// TIA Portal V16 export
// export: Created 2024-09-05T17:39:24.436191Z, ExportSetting WithDefaults, DisplayName Totally Integrated Automation Portal, DisplayVersion V16 Update 6, DisplayName TIA Portal Version Control Interface, DisplayVersion V16 Update 2, DisplayName TIA Portal Openness, DisplayVersion V16 Update 6, DisplayName STEP 7 Professional, DisplayVersion V16 Update 6, DisplayName STEP 7 Safety, DisplayVersion V16, DisplayName WinCC Advanced, DisplayVersion V16 Update 6
FUNCTION "Concatenate_STRING" : Void   // FC2010, LAD
{ S7_Optimized_Access := 'TRUE' }
VERSION : 0.1
// stored: AutoNumber false, IsIECCheckEnabled false, SetENOAutomatically false, UDAEnableTagReadback false
   VAR_INPUT
      DMC_SAP_REF : Array[1..10] of String[25];
   END_VAR
   VAR_OUTPUT
      String_empty : Bool;
   END_VAR
   VAR_IN_OUT
      DMC_SAP_REf_WSTRING : WString;
   END_VAR
   VAR_TEMP
      concatenate : String;
      Convert : WString;
   END_VAR
   VAR CONSTANT
      Template_string_empty : String := ';;;;;;;;;';
   END_VAR
BEGIN

REGION Network 1 (SCL): Concatenate function
       #concatenate := CONCAT(IN1 := #DMC_SAP_REF[1], IN2 := ';');
       #concatenate := CONCAT(IN1 := #concatenate, IN2 := #DMC_SAP_REF[2]);
       #concatenate := CONCAT(IN1 := #concatenate, IN2 := ';');
       #concatenate := CONCAT(IN1 := #concatenate, IN2 := #DMC_SAP_REF[3]);
       #concatenate := CONCAT(IN1 := #concatenate, IN2 := ';');
       #concatenate := CONCAT(IN1 := #concatenate, IN2 := #DMC_SAP_REF[4]);
       #concatenate := CONCAT(IN1 := #concatenate, IN2 := ';');
       #concatenate := CONCAT(IN1 := #concatenate, IN2 := #DMC_SAP_REF[5]);
       #concatenate := CONCAT(IN1 := #concatenate, IN2 := ';');
       #concatenate := CONCAT(IN1 := #concatenate, IN2 := #DMC_SAP_REF[6]);
       #concatenate := CONCAT(IN1 := #concatenate, IN2 := ';');
       #concatenate := CONCAT(IN1 := #concatenate, IN2 := #DMC_SAP_REF[7]);
       #concatenate := CONCAT(IN1 := #concatenate, IN2 := ';');
       #concatenate := CONCAT(IN1 := #concatenate, IN2 := #DMC_SAP_REF[8]);
       #concatenate := CONCAT(IN1 := #concatenate, IN2 := ';');
       #concatenate := CONCAT(IN1 := #concatenate, IN2 := #DMC_SAP_REF[9]);
       #concatenate := CONCAT(IN1 := #concatenate, IN2 := ';');
       #concatenate := CONCAT(IN1 := #concatenate, IN2 := #DMC_SAP_REF[10]);
END_REGION

REGION Network 2
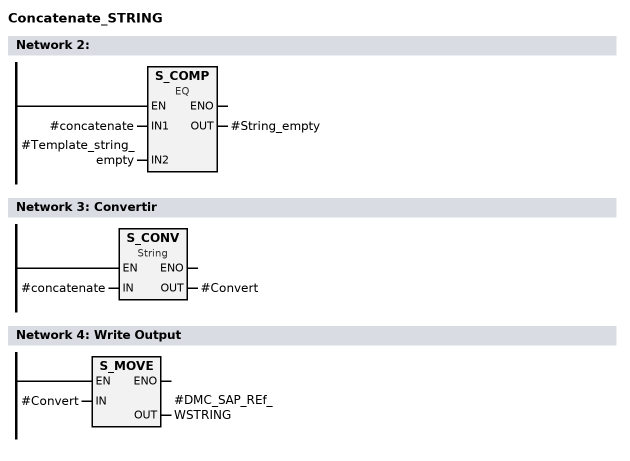
   RUNG wire#powerrail
      { S7_Templates := "[relation := EQ, src_type := String]" } S_COMP(IN1 := #concatenate, IN2 := #Template_string_empty, OUT => #String_empty)
   END_RUNG
   // the same network as SCL:
   S_COMP(IN1 := #concatenate, IN2 := #Template_string_empty, OUT => #String_empty);
END_REGION

REGION Network 3: Convertir
   RUNG wire#powerrail
      { S7_Templates := "[src_type := String, dest_type := WString]" } S_CONV(IN := #concatenate, OUT => #Convert)
   END_RUNG
   // the same network as SCL:
   S_CONV(IN := #concatenate, OUT => #Convert);
END_REGION

REGION Network 4: Write Output
   RUNG wire#powerrail
      S_Move(in := #Convert, out => #DMC_SAP_REf_WSTRING)
   END_RUNG
   // the same network as SCL:
   #DMC_SAP_REf_WSTRING := #Convert;
END_REGION
END_FUNCTION
